TYPE ST_CellConfig :
STRUCT
END_STRUCT
END_TYPE

(* stored: Version 1.1.0.1, ProductVersion 3.1.4024.12
   DUT ST_CellConfig: Id {b32367f4-9de0-4abd-bbd8-4550f4887423} *)
